// Simulation application main function
//
PROGRAM MAIN_SIMU
VAR

	// Function blocks...
	fbHeaterSimu: FB_HeaterSimu; // Heater simulation

	// Other members...
	Cntr: DINT; // Counter, visiting times
	
END_VAR

// Update counter
Cntr := ( Cntr + 1 );

// Call the heater simulation
fbHeaterSimu();

END_PROGRAM

(* stored: Version 1.1.0.1, ProductVersion 3.1.4022.6
   POU MAIN_SIMU: Id {be71b087-304f-4ff6-85a1-cb5aeb37af55}, SpecialFunc None *)
